# EPICS substitutions: epics/m-epics-eemcu/eemcuApp/Db/Sim8-extra-m8.substitutions
file "eemcu-extra.template"
{
pattern
{P,      M,    R,   PORT, ADDR, PREC, HOMEPROC}
{IOC:,   m8, m8-,   MCU1,    8, 3,    3}
}
